FUNCTION_BLOCK automaton
  (* Standard: 61499-2 *)
  (* Version 0.0, 2020-05-15, fbSAT, nxtControl GmbH *)
  PACKAGE Main;
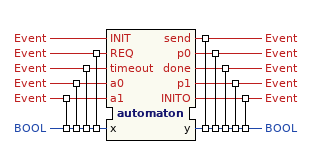
  EVENT_INPUT
    INIT;
    REQ WITH x;
    timeout WITH x;
    a0 WITH x;
    a1 WITH x;
  END_EVENT
  EVENT_OUTPUT
    send WITH y;
    p0 WITH y;
    done WITH y;
    p1 WITH y;
    INITO WITH y;
  END_EVENT
  VAR_INPUT
    x : BOOL;
  END_VAR
  VAR_OUTPUT
    y : BOOL;
  END_VAR
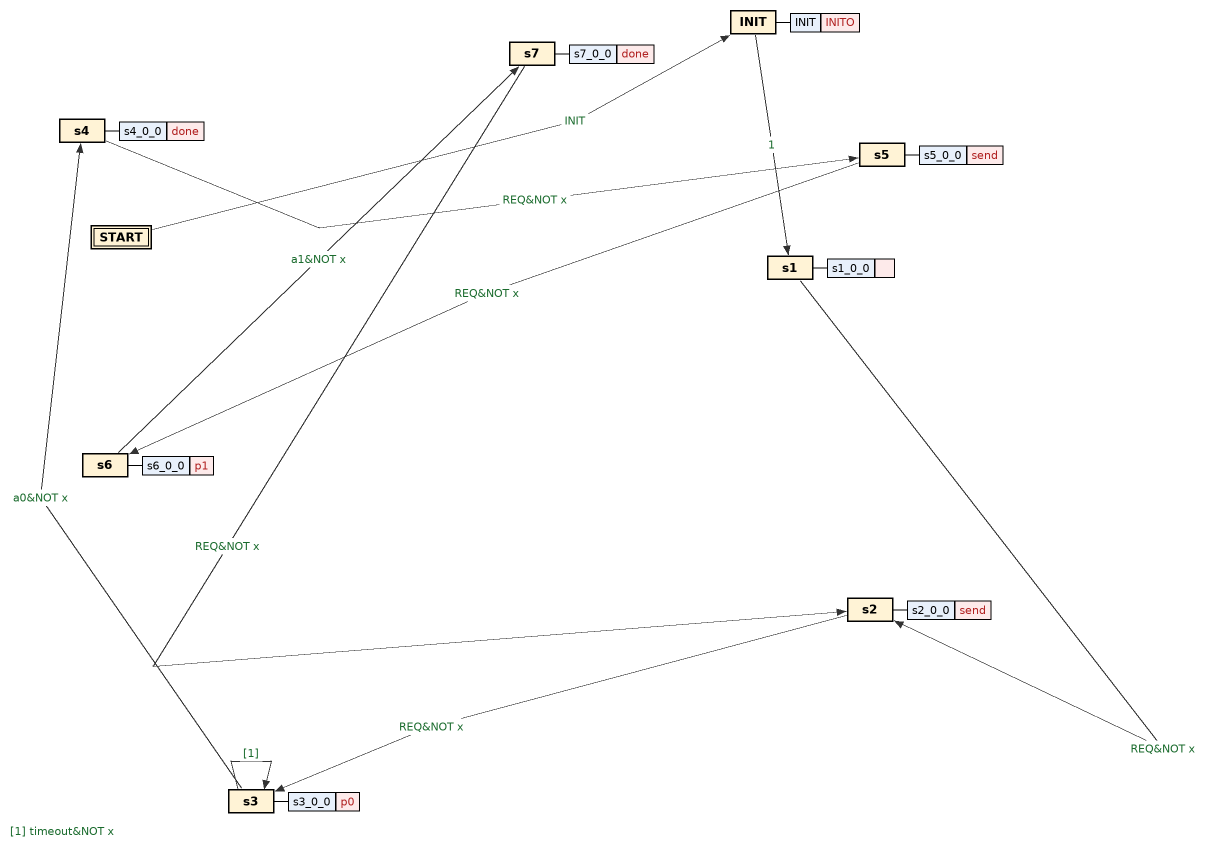
  EC_STATES
    START;
    INIT : INIT -> INITO;
    s1 : s1_0_0;
    s2 : s2_0_0 -> send;
    s3 : s3_0_0 -> p0;
    s4 : s4_0_0 -> done;
    s5 : s5_0_0 -> send;
    s6 : s6_0_0 -> p1;
    s7 : s7_0_0 -> done;
  END_STATES
  EC_TRANSITIONS
    START TO INIT := INIT;
    INIT TO s1 := 1;
    s1 TO s2 := REQ&NOT x;
    s2 TO s3 := REQ&NOT x;
    s3 TO s4 := a0&NOT x;
    s3 TO s3 := timeout&NOT x;
    s4 TO s5 := REQ&NOT x;
    s5 TO s6 := REQ&NOT x;
    s6 TO s7 := a1&NOT x;
    s7 TO s2 := REQ&NOT x;
  END_TRANSITIONS
  ALGORITHM INIT IN ST:
y:=FALSE;
  END_ALGORITHM
  ALGORITHM s2_0_0 IN ST:
y:=FALSE;
  END_ALGORITHM
  ALGORITHM s3_0_0 IN ST:
y:=FALSE;
  END_ALGORITHM
  ALGORITHM s4_0_0 IN ST:
y:=FALSE;
  END_ALGORITHM
  ALGORITHM s5_0_0 IN ST:
y:=FALSE;
  END_ALGORITHM
  ALGORITHM s6_0_0 IN ST:
y:=FALSE;
  END_ALGORITHM
  ALGORITHM s7_0_0 IN ST:
y:=FALSE;
  END_ALGORITHM
END_FUNCTION_BLOCK
